// TIA Portal V20 export
DATA_BLOCK "zFNet_10Child_DB_1"   // DB493
// stored: InstanceOfName CITI_Logic.zFNet_10Child, InstanceOfType FB, Namespace CITI_Logic
"CITI_Logic.zFNet_10Child"
   // VAR_INPUT
   //    IN_NumberOf_FN_Retries : Int;
   //    IN_Component_Quantity : Int;
   //    IN_FN_Response_FLT_Time : DInt;
   //    IN_OEM_Data : "CITI_Logic.FlexNet_Data";
   // END_VAR
   // VAR_OUTPUT
   //    FN_Data : "CITI_Logic.FlexNet_Data";
   //    FlexNet_White_Light : Bool;
   //    FlexNet_Green_Light : Bool;
   //    FlexNet_Buzzer : Bool;
   //    FlexNet_No_Response_Count : Int;
   //    FlexNet_DataReceivedByHost : Bool;
   //    FlexNet_Last_ResponseTime : DInt;
   // END_VAR
   // VAR
   //    FN_Dry_Cycle_Block : Bool;
   //    FN_OneShot : Array[1..32] of Bool;
   //    Clock_Data : DTL;
   //    System_Time_Tick : Time;
   //    Present_Time_Tick : Int;
   //    Previous_Time_Tick : Int;
   //    Difference_Time_Tick : Int;
   //    Difference_Time_DInt : DInt;
   //    TimerForFN_DataReady : DInt;
   //    TimerForFN_Response_Test : DInt;
   //    TimerFN_DataReady_Retry : DInt;
   //    TimerFN_BuzzerOn : DInt;
   //    FN_PUNDataRdy_Dly : Bool;
   //    FN_DataReady_Failed_Retry : Bool;
   //    FlasherOn : Bool;
   //    FN_NumberOf_Retries : Int;
   //    FN_Num_Of_Retry_Cnt_HMI : Int;
   //    FlexNet_Response_FLT_CNT : Int;
   //    TimerForFlasher : DInt;
   //    FN_Data_Recd_Delay : Bool;
   //    Timer_HQ_Delay : DInt;
   //    Timer_GreenLight_Delay : DInt;
   //    FN_Num_Of_Retries_CNT : Int;
   //    FlexNet_Part_Passed { ExternalAccessible := 'False'; ExternalVisible := 'False'; ExternalWritable := 'False'} : Bool;
   //    FlexNet_Part_Failed { ExternalAccessible := 'False'; ExternalVisible := 'False'; ExternalWritable := 'False'} : Bool;
   //    FlexNet_PassFail_Valid { ExternalAccessible := 'False'; ExternalVisible := 'False'; ExternalWritable := 'False'} : Bool;
   //    ON { ExternalAccessible := 'False'; ExternalVisible := 'False'; ExternalWritable := 'False'} : Bool;
   //    OFF { ExternalAccessible := 'False'; ExternalVisible := 'False'; ExternalWritable := 'False'} : Bool;
   //    ReadClock_Rslt { ExternalAccessible := 'False'; ExternalVisible := 'False'; ExternalWritable := 'False'} : Int;
   // END_VAR
BEGIN
END_DATA_BLOCK
